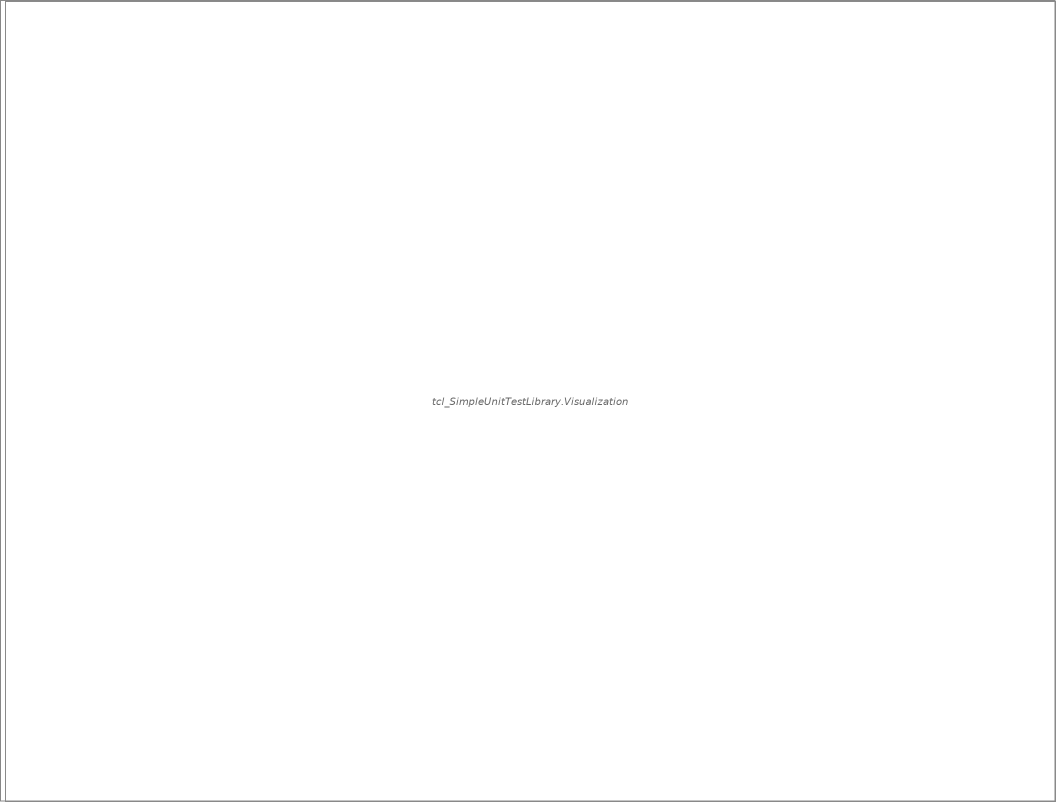
VISUALIZATION TestUI  // 1056x802
    Frame (5,1 1051x801)
        shows tcl_SimpleUnitTestLibrary.Visualization(TestRunner := PRG_Tests.testRunner)
END_VISUALIZATION

(* stored: Version 1.1.0.1, ProductVersion 3.1.4024.12
   Visu TestUI: Id {8a574625-3b20-4c0d-a46a-5c9d131d47b5} *)
